% RSLogix 500 project TRAFIC LIGHT CONTROLL FINAL PROGRMM_BAK006.RSS, saved by version 8.30.00.16 %
PROJECT "UNTITLED"    % processor: Bul.1763 MicroLogix 1100 Series B %

PROGRAM FILES
  LAD 2   20 rungs

DATA FILES
  O0 OUTPUT  4 elements
  I1 INPUT  6 elements
  S2 STATUS  66 elements
  B3 BINARY  1 elements
  T4 TIMER  10 elements
  C5 COUNTER  1 elements
  R6 CONTROL  1 elements
  N7 INTEGER  1 elements
  F8 FLOAT  1 elements

LADDER 2
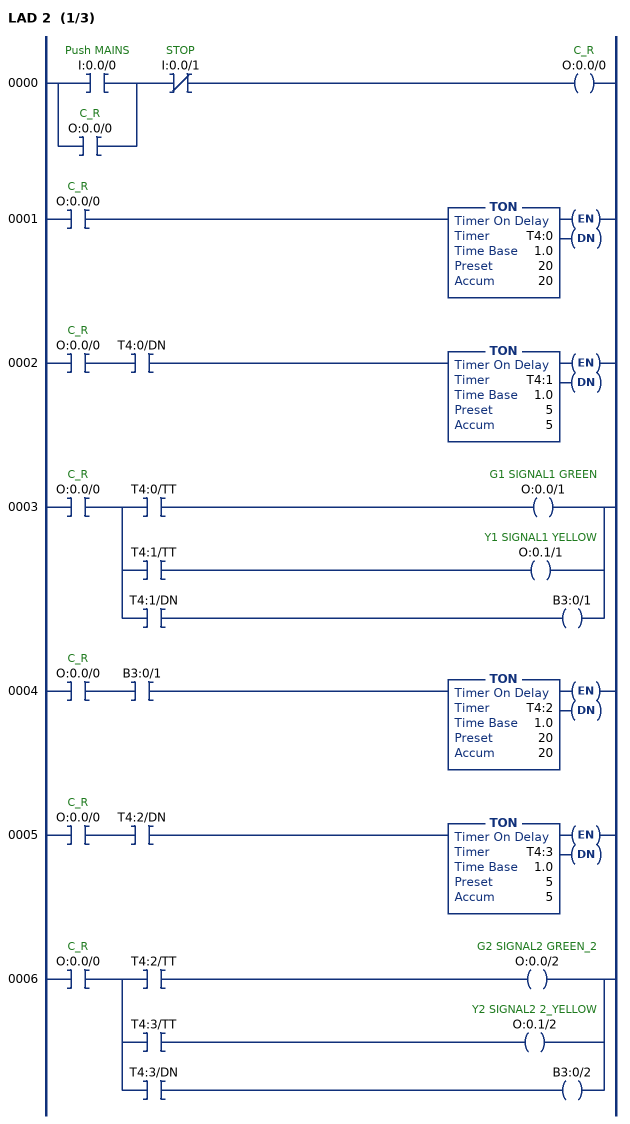
% Rung: 0 %
SOR BST XIC I:0.0/0 NXB XIC O:0.0/0 BND XIO I:0.0/1 OTE O:0.0/0 EOR
%   I:0.0/0  MAINS  "Push" %
%   O:0.0/0  C_R %
%   I:0.0/1  STOP %
% Rung: 1 %
SOR XIC O:0.0/0 TON T4:0 1.0 20 20 EOR
%   O:0.0/0  C_R %
% Rung: 2 %
SOR XIC O:0.0/0 XIC T4:0/DN TON T4:1 1.0 5 5 EOR
%   O:0.0/0  C_R %
% Rung: 3 %
SOR XIC O:0.0/0 BST XIC T4:0/TT OTE O:0.0/1 NXB XIC T4:1/TT OTE O:0.1/1 NXB XIC T4:1/DN OTE B3:0/1 BND EOR
%   O:0.0/0  C_R %
%   O:0.0/1  GREEN  "G1 SIGNAL1" %
%   O:0.1/1  YELLOW  "Y1 SIGNAL1" %
% Rung: 4 %
SOR XIC O:0.0/0 XIC B3:0/1 TON T4:2 1.0 20 20 EOR
%   O:0.0/0  C_R %
% Rung: 5 %
SOR XIC O:0.0/0 XIC T4:2/DN TON T4:3 1.0 5 5 EOR
%   O:0.0/0  C_R %
% Rung: 6 %
SOR XIC O:0.0/0 BST XIC T4:2/TT OTE O:0.0/2 NXB XIC T4:3/TT OTE O:0.1/2 NXB XIC T4:3/DN OTE B3:0/2 BND EOR
%   O:0.0/0  C_R %
%   O:0.0/2  GREEN_2  "G2 SIGNAL2" %
%   O:0.1/2  2_YELLOW  "Y2 SIGNAL2" %

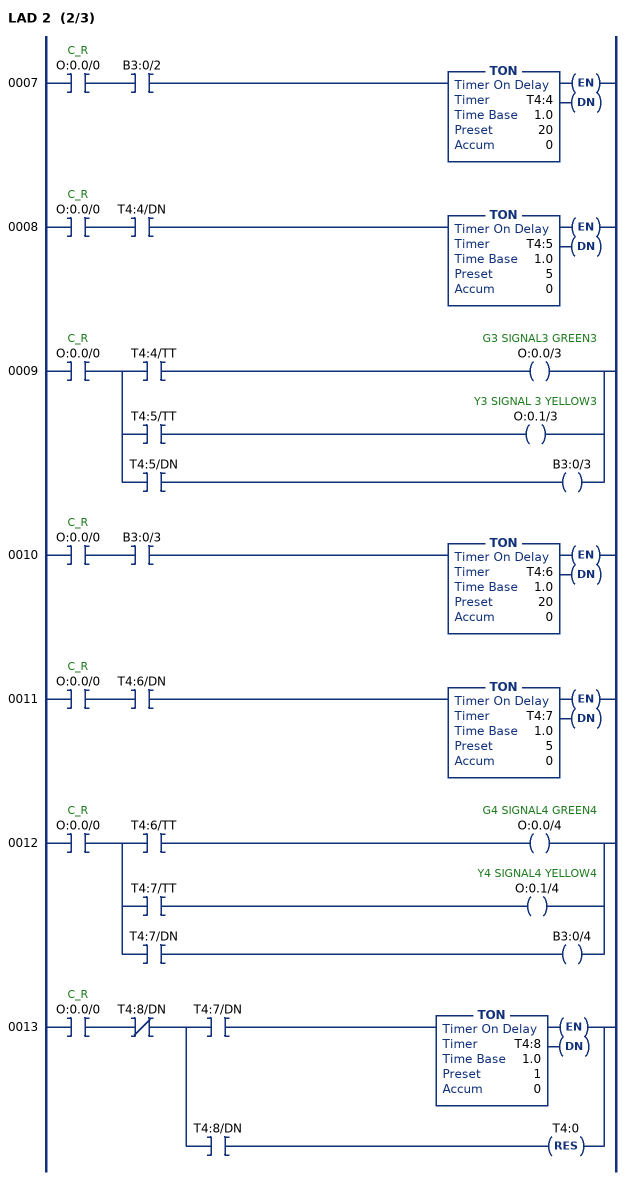
% Rung: 7 %
SOR XIC O:0.0/0 XIC B3:0/2 TON T4:4 1.0 20 0 EOR
%   O:0.0/0  C_R %
% Rung: 8 %
SOR XIC O:0.0/0 XIC T4:4/DN TON T4:5 1.0 5 0 EOR
%   O:0.0/0  C_R %
% Rung: 9 %
SOR XIC O:0.0/0 BST XIC T4:4/TT OTE O:0.0/3 NXB XIC T4:5/TT OTE O:0.1/3 NXB XIC T4:5/DN OTE B3:0/3 BND EOR
%   O:0.0/0  C_R %
%   O:0.0/3  GREEN3  "G3 SIGNAL3" %
%   O:0.1/3  YELLOW3  "Y3 SIGNAL 3" %
% Rung: 10 %
SOR XIC O:0.0/0 XIC B3:0/3 TON T4:6 1.0 20 0 EOR
%   O:0.0/0  C_R %
% Rung: 11 %
SOR XIC O:0.0/0 XIC T4:6/DN TON T4:7 1.0 5 0 EOR
%   O:0.0/0  C_R %
% Rung: 12 %
SOR XIC O:0.0/0 BST XIC T4:6/TT OTE O:0.0/4 NXB XIC T4:7/TT OTE O:0.1/4 NXB XIC T4:7/DN OTE B3:0/4 BND EOR
%   O:0.0/0  C_R %
%   O:0.0/4  GREEN4  "G4 SIGNAL4" %
%   O:0.1/4  YELLOW4  "Y4 SIGNAL4" %
% Rung: 13 %
SOR XIC O:0.0/0 XIO T4:8/DN BST XIC T4:7/DN TON T4:8 1.0 1 0 NXB XIC T4:8/DN RES T4:0 BND EOR
%   O:0.0/0  C_R %

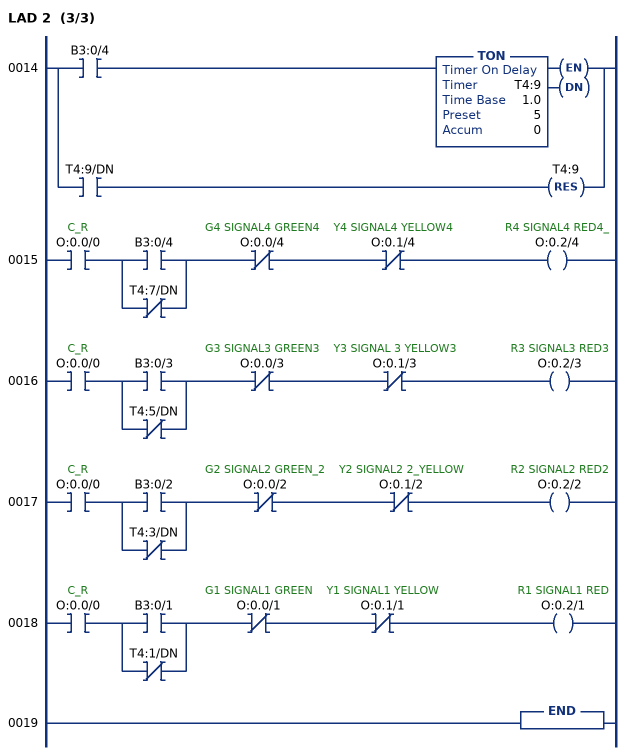
% Rung: 14 %
SOR BST XIC B3:0/4 TON T4:9 1.0 5 0 NXB XIC T4:9/DN RES T4:9 BND EOR
% Rung: 15 %
SOR XIC O:0.0/0 BST XIC B3:0/4 NXB XIO T4:7/DN BND XIO O:0.0/4 XIO O:0.1/4 OTE O:0.2/4 EOR
%   O:0.0/0  C_R %
%   O:0.0/4  GREEN4  "G4 SIGNAL4" %
%   O:0.1/4  YELLOW4  "Y4 SIGNAL4" %
%   O:0.2/4  RED4_  "R4 SIGNAL4" %
% Rung: 16 %
SOR XIC O:0.0/0 BST XIC B3:0/3 NXB XIO T4:5/DN BND XIO O:0.0/3 XIO O:0.1/3 OTE O:0.2/3 EOR
%   O:0.0/0  C_R %
%   O:0.0/3  GREEN3  "G3 SIGNAL3" %
%   O:0.1/3  YELLOW3  "Y3 SIGNAL 3" %
%   O:0.2/3  RED3  "R3 SIGNAL3" %
% Rung: 17 %
SOR XIC O:0.0/0 BST XIC B3:0/2 NXB XIO T4:3/DN BND XIO O:0.0/2 XIO O:0.1/2 OTE O:0.2/2 EOR
%   O:0.0/0  C_R %
%   O:0.0/2  GREEN_2  "G2 SIGNAL2" %
%   O:0.1/2  2_YELLOW  "Y2 SIGNAL2" %
%   O:0.2/2  RED2  "R2 SIGNAL2" %
% Rung: 18 %
SOR XIC O:0.0/0 BST XIC B3:0/1 NXB XIO T4:1/DN BND XIO O:0.0/1 XIO O:0.1/1 OTE O:0.2/1 EOR
%   O:0.0/0  C_R %
%   O:0.0/1  GREEN  "G1 SIGNAL1" %
%   O:0.1/1  YELLOW  "Y1 SIGNAL1" %
%   O:0.2/1  RED  "R1 SIGNAL1" %
% Rung: 19 %
SOR END EOR

DATA TABLE (non-zero values as saved)
DATA B3
% B3:0 % 0X0006
DATA T4
% .PRE .ACC %
% T4:0 % 20 20
% T4:1 % 5 5
% T4:2 % 20 20
% T4:3 % 5 5
% T4:4 % 20 0
% T4:5 % 5 0
% T4:6 % 20 0
% T4:7 % 5 0
% T4:8 % 1 0
% T4:9 % 5 0
